Fanuc KAREL source: EXP.kl

PROGRAM T
%NOLOCKGROUP
VAR
 v0 : REAL
 res : REAL
BEGIN
 res = EXP(v0)
END T
